// TIA Portal project "Lab01-git" (V16)

(* hardware
DEVICE "S7-1200 station_1"  S7-1200 Station
   slot 0: "Rack_0"  S7-1200 Rack  Rack  V1.0
   slot 1: "PLC_1"  CPU 1212C DC/DC/DC  6ES7 212-1AE40-0XB0  V4.4
*)

// ===== PLC "PLC_1"  CPU 1212C DC/DC/DC =====

VAR_GLOBAL   // PLC tag table "Default tag table"
   "System_Byte" AT %MB1 : Byte;
   "FirstScan" AT %M1.0 : Bool;
   "DiagStatusUpdate" AT %M1.1 : Bool;
   "AlwaysTRUE" AT %M1.2 : Bool;
   "AlwaysFALSE" AT %M1.3 : Bool;
   "Clock_Byte" AT %MB0 : Byte;
   "Clock_10Hz" AT %M0.0 : Bool;
   "Clock_5Hz" AT %M0.1 : Bool;
   "Clock_2.5Hz" AT %M0.2 : Bool;
   "Clock_2Hz" AT %M0.3 : Bool;
   "Clock_1.25Hz" AT %M0.4 : Bool;
   "Clock_1Hz" AT %M0.5 : Bool;
   "Clock_0.625Hz" AT %M0.6 : Bool;
   "Clock_0.5Hz" AT %M0.7 : Bool;
   "EntradaI0_0" AT %I0.0 : Bool;
   "SalidaQ0_0" AT %Q0.0 : Bool;
   "Marca2_0" AT %M2.0 : Bool;
END_VAR

FUNCTION "FC_Lab1" : Void   // FC1, LAD
{ S7_Optimized_Access := 'TRUE' }
VERSION : 0.1
   VAR_INPUT
      Entrada : Bool;
      Marca : Bool;
      Clock : Bool;
   END_VAR
   VAR_OUTPUT
      Salida : Bool;
   END_VAR
BEGIN

REGION Network 1
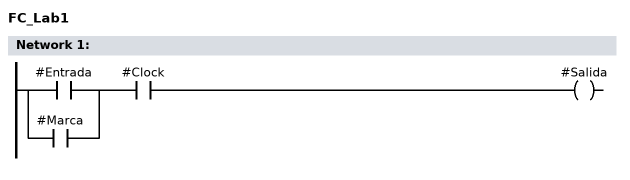
   RUNG wire#powerrail
      Contact( #Entrada )
      wire#w1
      Contact( #Clock )
      Coil( #Salida )
   END_RUNG
   RUNG wire#powerrail
      Contact( #Marca )
   END_RUNG wire#w1
   // the same network as SCL:
   #Salida := (#Entrada OR #Marca) AND #Clock;
END_REGION
END_FUNCTION

ORGANIZATION_BLOCK "Main"   // OB1, LAD, ProgramCycle
TITLE = "Main Program Sweep (Cycle)"
{ S7_Optimized_Access := 'TRUE' }
VERSION : 0.1
   VAR_INPUT
      Initial_Call : Bool;   // Initial call of this OB
      Remanence : Bool;   // =True, if remanent data are available
   END_VAR
BEGIN

REGION Network 1
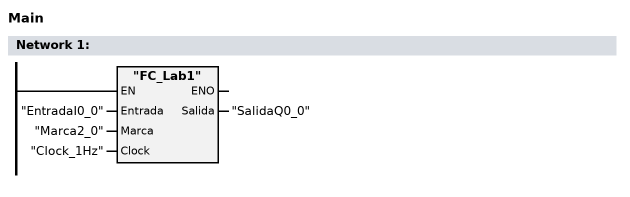
   RUNG wire#powerrail
      "FC_Lab1"(Entrada := "EntradaI0_0", Marca := "Marca2_0", Clock := "Clock_1Hz", Salida => "SalidaQ0_0")
   END_RUNG
   // the same network as SCL:
   "FC_Lab1"(Entrada := "EntradaI0_0", Marca := "Marca2_0", Clock := "Clock_1Hz", Salida => "SalidaQ0_0");
END_REGION
END_ORGANIZATION_BLOCK